(* CODESYS project Ladder1.project

Project tree, tasks and I/O mapping:
  Device : CODESYS Control Win V3, 3S - Smart Software Solutions GmbH, version 3.5.15.30
    application Application
      libraries: Standard, * (System)
      task MainTask (cyclic, interval t#20ms, priority 1) calls PLC_PRG [My first (Ladder) POU]
      task VISU_TASK (cyclic, interval 100 ms, priority 31) calls VisuElems.Visu_Prg
      program PLC_PRG [LD]
      visualisation Visualization1
  text list GlobalTextList
*)

// Device/Application/PLC_PRG
PROGRAM PLC_PRG
VAR
	Contact1: BOOL := FALSE;
	Coil1: BOOL;
	Contact2: BOOL := FALSE;
	Contact3: BOOL := TRUE;
END_VAR

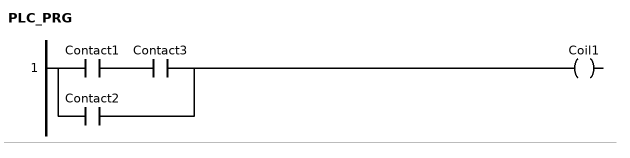
// NETWORK 1
Coil1 := Contact1 AND Contact3 OR Contact2;

END_PROGRAM

// Device/Application/Visualization1
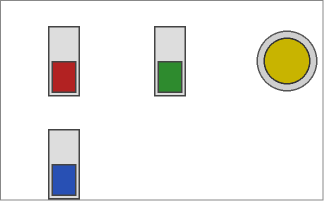
VISUALIZATION Visualization1  // 324x201
    DipSwitch (29,26 70x70), variable: PLC_PRG.Contact1, behaviour: TOGGLE, style: Switch-DipSwitch-Red
    Lamp1 (252,26 70x70), variable: PLC_PRG.Coil1, style: Lamp-Lamp1-Yellow
    DipSwitch (29,129 70x70), variable: PLC_PRG.Contact2, behaviour: TOGGLE, style: Switch-DipSwitch-Blue
    DipSwitch (135,26 70x70), variable: PLC_PRG.Contact3, behaviour: TOGGLE, style: Switch-DipSwitch-Green
END_VISUALIZATION
